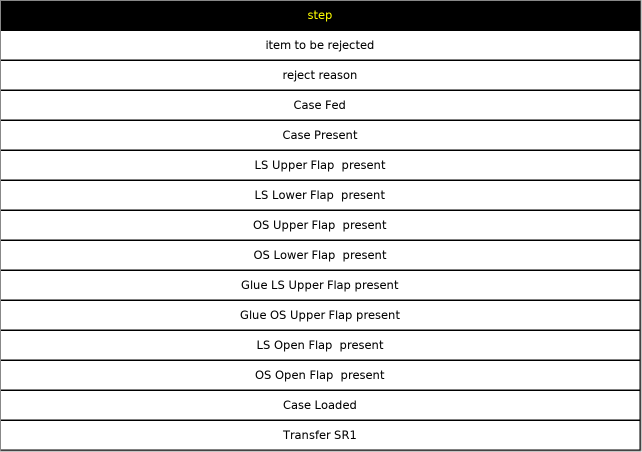
VISUALIZATION CUPS_FEEDING_SHIFT_ELEMENT_DESCRIPTION  // 642x452
    Rectangle (0,0 640x30), "step"
    Rectangle (0,30 640x30), "item to be rejected", tooltip "%d"
    Rectangle (0,60 640x30), "reject reason"
    Rectangle (0,90 640x30), "Case Fed"
    Rectangle (0,120 640x30), "Case Present"
    Rectangle (0,150 640x30), "LS Upper Flap present"
    Rectangle (0,180 640x30), "LS Lower Flap present"
    Rectangle (0,210 640x30), "OS Upper Flap present"
    Rectangle (0,240 640x30), "OS Lower Flap present"
    Rectangle (0,270 640x30), "Glue LS Upper Flap present"
    Rectangle (0,330 640x30), "LS Open Flap present"
    Rectangle (0,360 640x30), "OS Open Flap present"
    Rectangle (0,390 640x30), "Case Loaded"
    Rectangle (0,420 640x30), "Transfer SR1"
    Rectangle (0,300 640x30), "Glue OS Upper Flap present"
END_VISUALIZATION

(* stored: Version 1.1.0.1, ProductVersion 3.1.4024.3
   Visu CUPS_FEEDING_SHIFT_ELEMENT_DESCRIPTION: Id {d91b48d1-3e4a-42c6-936a-77536ec54731} *)
